{attribute 'linkalways'} 
{attribute 'no_explicit_call' := 'This FB is a CLASS and must be accessed using methods or properties'}
{attribute 'enable_dynamic_creation'}
FUNCTION_BLOCK _TcVnMatrix3x3_LREAL EXTENDS AliasDatatypeBase
VAR
	localData : TcVnMatrix3x3_LREAL;
	activeData : REFERENCE TO TcVnMatrix3x3_LREAL REF= localData;
	aliasBaseDatatype : _Array0to2_0to2OfLREAL;
END_VAR

PROPERTY PUBLIC Address : PVOID
GET
Address := ADR(activeData);
END_GET
END_PROPERTY

METHOD PUBLIC ClearReference
VAR_INPUT
END_VAR
activeData REF= localData;
SetBaseDatatypeReference();
END_METHOD

METHOD PUBLIC Clone : I_Datatype
VAR
    pClone : POINTER TO _TcVnMatrix3x3_LREAL;
END_VAR
pClone := __NEW(_TcVnMatrix3x3_LREAL);
Clone := pClone^;
END_METHOD

METHOD FB_init : BOOL
VAR_INPUT
	bInitRetains : BOOL; // if TRUE, the retain variables are initialized (warm start / cold start)
	bInCopyCode : BOOL;  // if TRUE, the instance afterwards gets moved into the copy code (online change)
	//InitialValue : TcVnMatrix3x3_LREAL; // if possible, not all values can be initialized
END_VAR
//localData := InitialValue; // if possible, not all values can be initialized
SetBaseDatatypeReference();
AddBaseDatatype(aliasBaseDatatype);
END_METHOD

PROPERTY PUBLIC Identifier : T_MAXSTRING
GET
Identifier := 'TcVnMatrix3x3_LREAL';
END_GET
END_PROPERTY

METHOD PUBLIC MakeReferenceTo
VAR_INPUT
	ReferenceTarget : REFERENCE TO TcVnMatrix3x3_LREAL;
END_VAR
activeData REF= ReferenceTarget;
SetBaseDatatypeReference();
END_METHOD

METHOD PROTECTED SetBaseDatatypeReference
VAR_INPUT
END_VAR
aliasBaseDatatype.MakeReferenceTo(activeData);
END_METHOD

PROPERTY PUBLIC Size : UDINT
GET
Size := SIZEOF(activeData);
END_GET
END_PROPERTY

METHOD TryMakeReferenceTo : BOOL
VAR_INPUT
	Target : I_Datatype;
END_VAR
VAR
	pTargetData : POINTER TO TcVnMatrix3x3_LREAL;
END_VAR
IF NOT IsEquivalentTo(Target) THEN
	RETURN;
END_IF

pTargetData := Target.Address;
activeData REF= pTargetData^;
SetBaseDatatypeReference();
TryMakeReferenceTo := TRUE;
END_METHOD

PROPERTY PUBLIC Value : REFERENCE TO TcVnMatrix3x3_LREAL
GET
Value REF= activeData;
END_GET
END_PROPERTY

END_FUNCTION_BLOCK

(* stored: Version 1.1.0.1, ProductVersion 3.1.4024.13
   POU _TcVnMatrix3x3_LREAL: Id {1b8a182f-bc5c-0538-3576-4989385b6ddd}, SpecialFunc None
   Folder Core: Id {0b259b4a-fccc-070d-0e4e-b59638dcabbd}
   Folder Protected: Id {12b1d4c6-8fb3-05ad-2d03-74552d732e4d}
   Folder Customize: Id {e63bda71-f819-002e-34a9-29aba297e695}
   Folder Constructor: Id {1f83ab9b-e33b-03c7-24e3-83ab9386e88f}
   Property Address: Id {fcb69f95-724b-096e-0175-8218be66ef28}
   Get Get: Id {57efe7af-9af4-0a1f-13ea-fdd2b68dcd1f}
   Method ClearReference: Id {aa947d4c-0ef9-076c-2653-c45ef3fea23a}
   Method Clone: Id {a2ffc7dc-f5c6-0acf-0116-b9b647440698}
   Method FB_init: Id {aaa3be17-c6c5-0813-261e-c35d27c93c85}
   Property Identifier: Id {7165728a-2db0-02b9-13ef-afbc9cc6c641}
   Get Get: Id {53fbd265-8bba-037e-325c-f15afe53b5fd}
   Method MakeReferenceTo: Id {4209f37e-f22e-0bfc-0ab6-73d189301404}
   Method SetBaseDatatypeReference: Id {d60fcce8-bc02-0264-1891-069d988d87ae}
   Property Size: Id {4f049f45-3815-0af8-205e-8ad8a701631d}
   Get Get: Id {3d8e0f04-b881-0159-1e3d-db70228bda84}
   Method TryMakeReferenceTo: Id {c26e85fd-37a8-0c8b-2f1d-fae45369ddf7}
   Property Value: Id {d3af85e2-0065-0e2e-295f-c62eb4e663b6}
   Get Get: Id {1f5610c9-3524-0c6d-05f9-90669ac11308} *)
